// TIA Portal V18 export
FUNCTION "SS2_IO_Update" : Void   // FC11100, LAD
{ S7_Optimized_Access := 'TRUE' }
VERSION : 0.1
// stored: AutoNumber false, IsIECCheckEnabled false, SetENOAutomatically false, UDAEnableTagReadback false
BEGIN

REGION Network 1
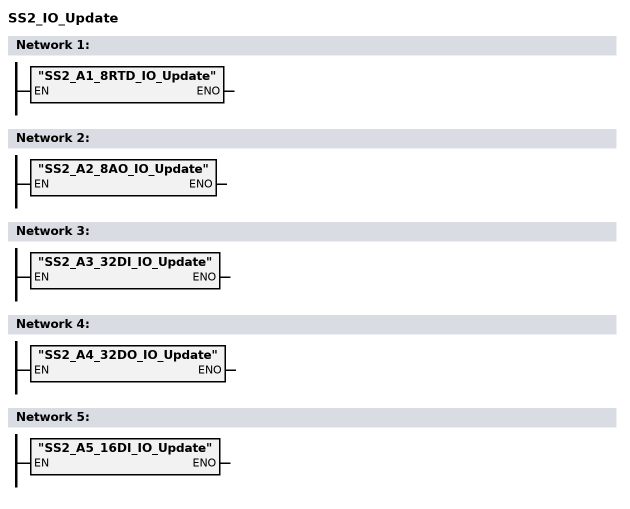
   RUNG wire#powerrail
      "SS2_A1_8RTD_IO_Update"()
   END_RUNG
   // the same network as SCL:
   "SS2_A1_8RTD_IO_Update"();
END_REGION

REGION Network 2
   RUNG wire#powerrail
      "SS2_A2_8AO_IO_Update"()
   END_RUNG
   // the same network as SCL:
   "SS2_A2_8AO_IO_Update"();
END_REGION

REGION Network 3
   RUNG wire#powerrail
      "SS2_A3_32DI_IO_Update"()
   END_RUNG
   // the same network as SCL:
   "SS2_A3_32DI_IO_Update"();
END_REGION

REGION Network 4
   RUNG wire#powerrail
      "SS2_A4_32DO_IO_Update"()
   END_RUNG
   // the same network as SCL:
   "SS2_A4_32DO_IO_Update"();
END_REGION

REGION Network 5
   RUNG wire#powerrail
      "SS2_A5_16DI_IO_Update"()
   END_RUNG
   // the same network as SCL:
   "SS2_A5_16DI_IO_Update"();
END_REGION
END_FUNCTION
